// Mitsubishi GX Works2 project: 5초 순서점등멸 신호등   PLC: Q00J

PROGRAM MAIN
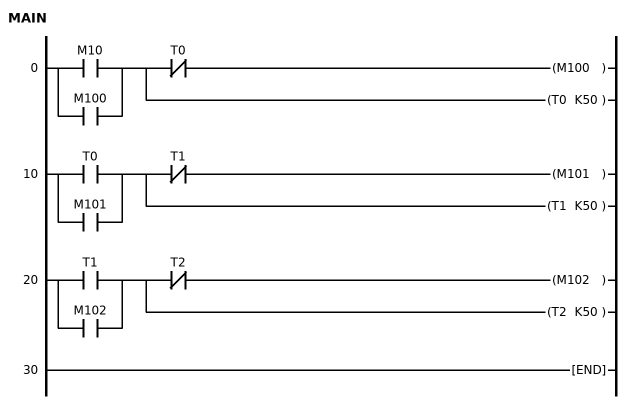
0     LD      M10
      OR      M100
      MPS
      ANI     T0
      OUT     M100
      MPP
      OUT     T0 K50
10    LD      T0
      OR      M101
      MPS
      ANI     T1
      OUT     M101
      MPP
      OUT     T1 K50
20    LD      T1
      OR      M102
      MPS
      ANI     T2
      OUT     M102
      MPP
      OUT     T2 K50
30    END
END_PROGRAM
